                ELSIF bPendingOperatorResultPass THEN

                    sMachineMessage :=
                        'Remove passed part from operator nest';

                ELSE

                    sMachineMessage :=
                        'Remove processed part from operator nest';

                END_IF


            // =================================================================
            E_OperatorExchangeState.WaitingForRejectConfirmation:
            // =================================================================

                // This state is reached only after removal has been confirmed.
                // Do not show a "confirmed" message here. Once the reject pulse
                // is accepted, the state machine exits this state automatically.
                sMachineMessage :=
                    'Place failed part in reject station';


            // =================================================================
            E_OperatorExchangeState.WaitingForPuckRemoval:
            // =================================================================

                IF bPuckLockerEnabled THEN

                    IF GVL_MASTER.stPuckLocker.bPuckDetected THEN

                        sMachineMessage :=
                            'Remove released puck from locker';

                    ELSE

                        sMachineMessage :=
                            'Insert new puck into locker';

                    END_IF

                ELSE

                    // Recovery protection if the locker is disabled while
                    // this state is still active.
                    sMachineMessage :=
                        'Completing operator exchange';

                END_IF


            // =================================================================
            E_OperatorExchangeState.WaitingForNewPuck:
            // =================================================================

                IF bPuckLockerEnabled THEN

                    sMachineMessage :=
                        'Insert new puck into locker';

                ELSE

                    sMachineMessage :=
                        'Completing operator exchange';

                END_IF


            // =================================================================
            E_OperatorExchangeState.WaitingForPuckLocked:
            // =================================================================

                IF bPuckLockerEnabled THEN

                    sMachineMessage :=
                        'Waiting for puck locker to lock';

                ELSE

                    sMachineMessage :=
                        'Completing operator exchange';

                END_IF


            // =================================================================
            E_OperatorExchangeState.WaitingForPartLoading:
            // =================================================================

                IF GVL_MASTER.stSensors.bPartPresent_NEST THEN

                    sMachineMessage :=
                        'Part loaded - ready to index';

                ELSE

                    sMachineMessage :=
                        'Load new part into operator nest';

                END_IF


            // =================================================================
            E_OperatorExchangeState.ExchangeComplete:
            // =================================================================

                sMachineMessage :=
                    'Operator exchange complete - press both safety controls to index';


            // =================================================================
            E_OperatorExchangeState.WaitingForTableIndexComplete:
            // =================================================================

                // Normally table movement is caught by the higher-priority
                // bNestInMotion condition. This message covers the transition
                // immediately before or after physical movement.
                sMachineMessage :=
                    'Index table moving - keep hands clear';


            // =================================================================
            ELSE
            // =================================================================

                sMachineMessage := '';

        END_CASE

    END_IF

END_IF


// -----------------------------------------------------------------------------
// Publish current machine instruction.
// -----------------------------------------------------------------------------
GVL_MASTER.sMachineMessage :=
    sMachineMessage;


// -----------------------------------------------------------------------------
// Temporary direct connection to DataGrid row zero.
// -----------------------------------------------------------------------------
GVL_MASTER.astActiveEvents[0].sEventTex :=
    sMachineMessage;

GVL_MASTER.astActiveEvents[0].sType :=
    'Message';

GVL_MASTER.astActiveEvents[0].sSolution :=
    '';

GVL_MASTER.astActiveEvents[0].abType :=
    3;
END_METHOD

METHOD PRIVATE M_UpdateOperatorInstruction
VAR_INPUT
END_VAR
END_METHOD

METHOD PRIVATE M_UpdateOperatorNestTracking
VAR
	iOperatorNestIndex 	: INT;
    iNest               : INT;
    bPartPresent        : BOOL;
END_VAR
// Pulses are valid for one PLC scan only.
// Clear all previous events before evaluating the current operator nest.
FOR iNest := 1 TO 4 DO

    GVL_MASTER.astNestTracking[iNest].bPartRemovedPulse := FALSE;
    GVL_MASTER.astNestTracking[iNest].bPartLoadedPulse := FALSE;

END_FOR

// Track the operator sensor while the table is safely stationary.
// IDLE is required for the initial loading sequence.
// TESTING is required for the normal unload/reload sequence.
IF (
        eNestState <> E_NestState.IDLE
        AND eNestState <> E_NestState.TESTING
        AND eNestState <> E_NestState.WAIT_OPERATOR_EXCHANGE
   )
   OR GVL_MASTER.stNestTable.bNestInMotion
   OR NOT GVL_MASTER.stNestTable.bNestReadySensor
   OR NOT GVL_MASTER.stNestTable.bNestLockedSensor
   OR eOperatorNestPosition = E_NestPosition.Unknown THEN

    RETURN;

END_IF

// E_NestPosition corresponds to indexes 1..4.
iOperatorNestIndex := TO_INT(eOperatorNestPosition);

IF (iOperatorNestIndex < 1) OR (iOperatorNestIndex > 4) THEN
    RETURN;
END_IF

// The physical sensor represents the nest currently accessible
// to the operator.
bPartPresent := GVL_MASTER.stSensors.bPartPresent_NEST;

// Detect a part placed into a disabled nest at the operator position.
// The condition follows the physical sensor directly so it clears
// automatically when the operator removes the part.
bDisabledNestPartPresent :=
    NOT M_IsNestEnabled(eOperatorNestPosition)
    AND bPartPresent;
// ============================================================================
// PART REMOVAL CONTROL WITHOUT PUCK LOCKER
// ============================================================================

// Evaluate the part sensor only when a different nest has arrived
// at the operator position.
//
// A part already present when the nest arrives is considered a processed
// part and must be removed before the table can index again.
IF GVL_HMI.stPuckLocker.eMode = E_PuckLockerMode.Disabled THEN

    IF eOperatorNestPosition <> eLastOperatorNestPositionNoLocker THEN

        eLastOperatorNestPositionNoLocker := eOperatorNestPosition;

        bPartRemovalRequiredNoLocker := bPartPresent;

    END_IF

ELSE

    // This memory is not used when the Puck Locker is enabled.
    bPartRemovalRequiredNoLocker := FALSE;

    // Keep the current position synchronized so that changing modes does
    // not create a false new-position detection.
    eLastOperatorNestPositionNoLocker := eOperatorNestPosition;

END_IF

// Detect processed part removal.
GVL_MASTER.astNestTracking[iOperatorNestIndex].bPartRemovedPulse := GVL_MASTER.astNestTracking[iOperatorNestIndex].bPreviousSensor AND NOT bPartPresent;

// Once the part that arrived with the nest has been physically removed,
// allow the next index.
//
// Loading another part afterwards must not reactivate this requirement.
IF GVL_HMI.stPuckLocker.eMode = E_PuckLockerMode.Disabled
   AND bPartRemovalRequiredNoLocker
   AND GVL_MASTER.astNestTracking[iOperatorNestIndex].bPartRemovedPulse THEN

    bPartRemovalRequiredNoLocker := FALSE;

END_IF

// Detect new part loading.
GVL_MASTER.astNestTracking[iOperatorNestIndex].bPartLoadedPulse :=
    NOT GVL_MASTER.astNestTracking[iOperatorNestIndex].bPreviousSensor
    AND bPartPresent;

// Retain the logical occupancy of this physical nest.
//
// The physical sensor is only available at the operator position.
// Therefore, bPartLoaded must represent the remembered part state
// associated with the nest, not a continuous copy of the sensor.
IF GVL_MASTER.astNestTracking[iOperatorNestIndex].bPartLoadedPulse THEN

    // A new physical part has been loaded into this nest.
    GVL_MASTER.astNestTracking[iOperatorNestIndex].bPartLoaded := TRUE;

    // A new part must never inherit the process result
    // stored for the previous part in the same physical nest.
    GVL_MASTER.astNestProcessResult[iOperatorNestIndex].bResultValid := FALSE;
    GVL_MASTER.astNestProcessResult[iOperatorNestIndex].bPass := FALSE;
    GVL_MASTER.astNestProcessResult[iOperatorNestIndex].bFail := FALSE;
    GVL_MASTER.astNestProcessResult[iOperatorNestIndex].bDispositionSent := FALSE;

ELSIF GVL_MASTER.astNestTracking[iOperatorNestIndex].bPartRemovedPulse THEN

    GVL_MASTER.astNestTracking[iOperatorNestIndex].bPartLoaded := FALSE;

END_IF

// Save the current sensor state for the next scan.
GVL_MASTER.astNestTracking[iOperatorNestIndex].bPreviousSensor :=
    bPartPresent;
END_METHOD

METHOD PRIVATE M_UpdatePuckLockerPartRemovalStatus
VAR
	iOperatorNestIndex : INT;
END_VAR
// Keep the removal confirmation active until the Puck Locker
// acknowledges it by leaving the Locked state.
//
// Do not forward the one-scan physical sensor pulse directly.
GVL_MASTER.stPuckLocker.bPartRemovedFromNest := bPendingOperatorResultPass AND bPartRemovedConfirmedForExchange;
END_METHOD

METHOD PRIVATE M_UpdatePuckLockerPermissives
VAR_INPUT
END_VAR
// Puck Locker is considered permissive when disabled,
// or when enabled without any latched locker fault.
GVL_MASTER.stPuckLocker.bMachinePermissive :=
    (GVL_HMI.stPuckLocker.eMode = E_PuckLockerMode.Disabled)
    OR
    (
        NOT GVL_MASTER.stPuckLocker.bUnexpectedRemovalFault
        AND NOT GVL_MASTER.stPuckLocker.bPuckSensorMismatch
        AND GVL_MASTER.stPuckLocker.eState
            <> E_PuckLockerState.UnexpectedPuckRemovalFault
    );


// The table can index only after the complete operator-exchange
// sequence has finished.
//
// PASS:
// Part removed from nest -> exchange complete.
//
// FAIL:
// Part removed from nest -> reject sensor confirmed
// -> exchange complete.
GVL_MASTER.stPuckLocker.bIndexPermissive :=
    GVL_MASTER.stPuckLocker.bMachinePermissive
    AND bOperatorExchangeComplete
	AND NOT bDisabledNestPartPresent;
END_METHOD

METHOD M_UpdateStatisticsAndHistory
VAR_INPUT
END_VAR
// =========================================================
// LOCAL SYSTEM TIME
// =========================================================

// Update the local system time cyclically.
fbLocalSystemTime(
    bEnable := TRUE,
    dwCycle := 1
);


// =========================================================
// DATA HISTORY INDEX VALIDATION
// =========================================================

IF (GVL_HMI.iDataHistoryWriteIndex < 1)
   OR (GVL_HMI.iDataHistoryWriteIndex > 2000) THEN

    GVL_HMI.iDataHistoryWriteIndex := 1;

END_IF


// =========================================================
// DETECT FINAL STORED KISTLER RESULT
// =========================================================

// Generate a one-cycle pulse only after the final AutoCycle
// Kistler result has been stored in aKistlerNestResult.
rtKistlerResultDone(
    CLK := bKistlerResultStored
);


// Only automatic production results are allowed to update
// Statistics, Data History and CSV.
IF rtKistlerResultDone.Q
   AND GVL_MASTER.stMachineStatus.eMachineState =
       E_MachineState.SYSTEM_AUTO_CYCLE THEN


    // =====================================================
    // SAFE NEST POSITION MAPPING
    // =====================================================

    CASE eCurrentNestPos OF

        E_NestPosition.Position_1:
            iDataHistoryNestIndex := 1;

        E_NestPosition.Position_2:
            iDataHistoryNestIndex := 2;

        E_NestPosition.Position_3:
            iDataHistoryNestIndex := 3;

        E_NestPosition.Position_4:
            iDataHistoryNestIndex := 4;

    ELSE

        iDataHistoryNestIndex := 0;

    END_CASE


    // =====================================================
    // STATISTICS
    // =====================================================

    // Update statistics only when the nest position is valid.
    IF (iDataHistoryNestIndex >= 1)
       AND (iDataHistoryNestIndex <= 4) THEN

        IF stKistler_Status.bPartOK THEN

            // Total machine statistics.
            GVL_HMI.udiKistlerTotalTested :=
                GVL_HMI.udiKistlerTotalTested + 1;

            GVL_HMI.udiKistlerTotalPass :=
                GVL_HMI.udiKistlerTotalPass + 1;

            // Good parts for this nest.
            GVL_HMI.aKistlerNestGoodParts[
                iDataHistoryNestIndex
            ] :=
                GVL_HMI.aKistlerNestGoodParts[
                    iDataHistoryNestIndex
                ] + 1;


        ELSIF stKistler_Status.bPartNOK THEN

            // Total machine statistics.
            GVL_HMI.udiKistlerTotalTested :=
                GVL_HMI.udiKistlerTotalTested + 1;

            GVL_HMI.udiKistlerTotalFail :=
                GVL_HMI.udiKistlerTotalFail + 1;

            // Bad parts for this nest.
            GVL_HMI.aKistlerNestBadParts[
                iDataHistoryNestIndex
            ] :=
                GVL_HMI.aKistlerNestBadParts[
                    iDataHistoryNestIndex
                ] + 1;

        END_IF


        // =====================================================
        // STORE DATA HISTORY ENTRY
        // =====================================================

        // Nest.
        GVL_HMI.aDataHistoryHMI[
            GVL_HMI.iDataHistoryWriteIndex
        ].iNestIndex :=
            iDataHistoryNestIndex;


        // Result.
        IF stKistler_Status.bPartOK THEN

            GVL_HMI.aDataHistoryHMI[
                GVL_HMI.iDataHistoryWriteIndex
            ].sResult := 'PASS';

        ELSIF stKistler_Status.bPartNOK THEN

            GVL_HMI.aDataHistoryHMI[
                GVL_HMI.iDataHistoryWriteIndex
            ].sResult := 'FAIL';

        ELSE

            GVL_HMI.aDataHistoryHMI[
                GVL_HMI.iDataHistoryWriteIndex
            ].sResult := '';

        END_IF


        // Force.
        // Use the final value already stored for this nest.
        GVL_HMI.aDataHistoryHMI[
            GVL_HMI.iDataHistoryWriteIndex
        ].rForce :=
            GVL_HMI.aKistlerNestResult[
                iDataHistoryNestIndex
            ].rForce;


        // Distance.
        // Use the final value already stored for this nest.
        GVL_HMI.aDataHistoryHMI[
            GVL_HMI.iDataHistoryWriteIndex
        ].rDistance :=
            GVL_HMI.aKistlerNestResult[
                iDataHistoryNestIndex
            ].rDistance;


        // Date and time.
        GVL_HMI.aDataHistoryHMI[
            GVL_HMI.iDataHistoryWriteIndex
        ].dtTimeStamp :=
            SYSTEMTIME_TO_DT(
                fbLocalSystemTime.systemTime
            );


        // =====================================================
        // PREPARE CSV DATA
        // =====================================================

        // Copy the complete Data History record before moving
        // the circular buffer index.
        GVL_HMI.stCSVDataPending :=
            GVL_HMI.aDataHistoryHMI[
                GVL_HMI.iDataHistoryWriteIndex
            ];

        // Request CSV storage for this completed Kistler test.
        GVL_HMI.bCSVWriteRequest := TRUE;


        // Move to the next history position.
        GVL_HMI.iDataHistoryWriteIndex :=
            GVL_HMI.iDataHistoryWriteIndex + 1;


        // Circular history.
        IF GVL_HMI.iDataHistoryWriteIndex > 2000 THEN

            GVL_HMI.iDataHistoryWriteIndex := 1;

        END_IF

    END_IF

END_IF


// =========================================================
// HMI STATISTICS MAPPING
// =========================================================

GVL_HMI.aStatisticsHMI[1].udiTotalTested :=
    GVL_HMI.udiKistlerTotalTested;

GVL_HMI.aStatisticsHMI[1].udiGoodParts :=
    GVL_HMI.udiKistlerTotalPass;

GVL_HMI.aStatisticsHMI[1].udiBadParts :=
    GVL_HMI.udiKistlerTotalFail;


// Calculate efficiency.
IF GVL_HMI.aStatisticsHMI[1].udiTotalTested > 0 THEN

    GVL_HMI.aStatisticsHMI[1].rEfficiency :=
        UDINT_TO_REAL(
            GVL_HMI.aStatisticsHMI[1].udiGoodParts
        )
        * 100.0
        /
        UDINT_TO_REAL(
            GVL_HMI.aStatisticsHMI[1].udiTotalTested
        );

ELSE

    GVL_HMI.aStatisticsHMI[1].rEfficiency := 0.0;

END_IF


// =========================================================
// RESET STATISTICS ONLY
// =========================================================

IF GVL_HMI.aStatisticsHMI[1].bReset THEN

    // Reset total machine statistics.
    GVL_HMI.udiKistlerTotalTested := 0;
    GVL_HMI.udiKistlerTotalPass := 0;
    GVL_HMI.udiKistlerTotalFail := 0;

    // Reset per-nest statistics.
    GVL_HMI.aKistlerNestGoodParts[1] := 0;
    GVL_HMI.aKistlerNestGoodParts[2] := 0;
    GVL_HMI.aKistlerNestGoodParts[3] := 0;
    GVL_HMI.aKistlerNestGoodParts[4] := 0;

    GVL_HMI.aKistlerNestBadParts[1] := 0;
    GVL_HMI.aKistlerNestBadParts[2] := 0;
    GVL_HMI.aKistlerNestBadParts[3] := 0;
    GVL_HMI.aKistlerNestBadParts[4] := 0;

    // Do not clear aDataHistoryHMI.
    // Do not reset iDataHistoryWriteIndex.

    // Clear the HMI request.
    GVL_HMI.aStatisticsHMI[1].bReset := FALSE;

END_IF


// =========================================================
// CLEAR ONE HISTORY ENTRY PER PLC CYCLE
// =========================================================

// Clearing one entry per scan avoids processing all 2000
// structures in a single PLC cycle.
// IF bDataHistoryResetActive THEN
//
//     GVL_HMI.aDataHistoryHMI[
//         iDataHistoryResetIndex
//     ].iNestIndex := 0;
//
//     GVL_HMI.aDataHistoryHMI[
//         iDataHistoryResetIndex
//     ].sResult := '';
//
//     GVL_HMI.aDataHistoryHMI[
//         iDataHistoryResetIndex
//     ].rDistance := 0.0;
//
//     GVL_HMI.aDataHistoryHMI[
//         iDataHistoryResetIndex
//     ].rForce := 0.0;
//
//     GVL_HMI.aDataHistoryHMI[
//         iDataHistoryResetIndex
//     ].dtTimeStamp :=
//         DT#1970-01-01-00:00:00;
//
//
//     IF iDataHistoryResetIndex < 2000 THEN
//
//         iDataHistoryResetIndex :=
//             iDataHistoryResetIndex + 1;
//
//     ELSE
//
//         // History clearing completed.
//         GVL_HMI.iDataHistoryWriteIndex := 1;
//
//         iDataHistoryResetIndex := 1;
//         bDataHistoryResetActive := FALSE;
//
//     END_IF
//
// END_IF
END_METHOD

END_PROGRAM

(* stored: Version 1.1.0.1
   POU PRG_MachineControl: Id {73cce6c0-0336-454e-b089-fed285c9fc85}, SpecialFunc None
   Folder GuideCylinder: Id {f10faf9c-65dc-4eb4-9dd1-2b0b5aecf204}
   Folder Kistler: Id {9e17cfcd-c98c-45cb-bd0b-324e8c0aff3a}
   Folder Nest_Table: Id {b7ca633f-afa1-44ec-8055-793fa5c0679e}
   Folder Pick_Locker: Id {df051fcd-8c9f-4620-b035-4bdfd7cf7977}
   Folder SupportElevator: Id {7f702417-a10d-4779-8751-86ff4b21f60e}
   Method M_ClearCompletedOperatorNestResult: Id {01b8ae27-8d16-43ef-a386-7432c49082ed}
   Method M_ClearRemovedOperatorNestResult: Id {c718cf76-b546-4927-a46e-0e5025b89a81}
   Method M_ConfirmPuckLockerDisposition: Id {10b0db97-52e9-4e62-9b4d-4520c43ca38e}
   Method M_GetCurrentPosition: Id {5ad458d2-2562-4615-8d3c-a8c74f1cf84a}
   Method M_GuideCylinderControl: Id {104c92f2-fa5c-4064-a20d-a8f4a2c78ac7}
   Method M_HMIKistlerResult: Id {5ec231b7-f8ff-4c60-8cb2-2f6710f94bba}
   Method M_IsNestEnabled: Id {faec0923-f0a4-4b40-99ae-0b504fd30bb5}
   Method M_KistlerCommandMapping: Id {5cfa21d9-3cc5-49b3-924c-97638c44a598}
   Method M_KistlerConfig_Input: Id {14c376fa-cf59-47d0-a1ae-92a997aeb833}
   Method M_KistlerConfig_Output: Id {8ae5f917-1437-4f6b-8e62-9b5bec1a92a3}
   Method M_KistlerControl: Id {142f0c7b-5ff7-4bb2-a407-a7b85664501f}
   Method M_KistlerStateMachine: Id {537fbedf-c4eb-4029-b5fd-b3d3431bc3e9}
   Method M_LEDsButtons: Id {a6680c49-408d-47a5-bfa3-499d1bfac7ad}
   Method M_NestTableControl: Id {73045679-2a70-4e2a-a7bb-96539b2fce6a}
   Method M_OperatorExchangeControl: Id {531cdfdc-4414-409e-a0f2-21c7605d741a}
   Method M_PreExecution: Id {d5c5735d-f733-481f-9f83-00134f7ccc98}
   Method M_ProcessCycle: Id {e01c53ef-c471-4f56-958b-74875adab0b2}
   Method M_PuckLockerDisposition: Id {ad617b9e-72f0-4e71-8779-255d6dead4ac}
   Method M_ResetProcessCycle: Id {454cd463-1fae-4730-b15d-6fd1047cb008}
   Method M_StartFaultRejectRecovery: Id {1379298e-0cfb-4338-ae73-185b8119dc5c}
   Method M_StatusMapping: Id {e76387c3-2b6b-4ab8-8e2c-031286cbd112}
   Method M_StoreKistlerResult: Id {44a9f0cc-607f-440e-a240-216b02f970e5}
   Method M_SupportControl: Id {64d76664-69d4-4214-9755-744a37e12132}
   Method M_TerminalInfo: Id {3b4d5e27-92fa-407f-953a-0393950625d4}
   Method M_UpdateActiveNestPositions: Id {a175beaf-3ad8-4d7b-8c4f-5074246f2c65}
   Method M_UpdateMachineMessage: Id {be75d2f8-1d8e-4982-923d-f25114b7d3b4}
   Method M_UpdateOperatorInstruction: Id {9003e453-721d-4c1e-a060-193bc77fe83e}
   Method M_UpdateOperatorNestTracking: Id {d4e87f72-d62a-4a59-bdf7-747a3fa48afb}
   Method M_UpdatePuckLockerPartRemovalStatus: Id {f9bf3ed2-647f-49ac-acef-7d7719e93b2e}
   Method M_UpdatePuckLockerPermissives: Id {a5082c5a-ff24-4e5c-a334-ef2912094065}
   Method M_UpdateStatisticsAndHistory: Id {00ee633c-8762-44a1-a124-fd33218f5608} *)
